(* CoDeSys 2.3 export: ROUNDINGTO5.EXP *)

(* POU 05_Basic_Calc/roundingTo5, ST *)
FUNCTION roundingTo5 : UINT 	(* Функция окргуляет число до ближайшего кратного (5 * order) числа *)
VAR_INPUT
	in_number_u16	: UINT;		(* Число, которое нужно округлить *)
	order				: UINT;		(* Порядок до которого округлять. 1 – до кратного 5ти, 10 – до кратного 50ти, и тд... *)
END_VAR
VAR
	div_part			: REAL;		(* Целое число *)
	aux_num			: UINT;		(* вспомогательная переменная для отслеживания округления до меньшего целого *)
	dec_part			: REAL;		(* десятая часть числа *)
END_VAR
VAR CONSTANT
	LOW_ROUND		: REAL := 0.25;
	HIGH_ROUND		: REAL := 0.75;
END_VAR
IF order < 1 THEN
	roundingTo5 := in_number_u16;
ELSE
	IF order < 10 THEN
		order := 1;
	ELSIF order < 100 THEN
		order := 10;
	ELSIF order < 1000 THEN
		order := 100;
	ELSIF order < 10000 THEN
		order := 1000;
	ELSE
		order := 10000;
	END_IF

	div_part	:= UINT_TO_REAL(in_number_u16) / (order * 10);
	aux_num	:= REAL_TO_UINT(div_part);
	
	IF UINT_TO_REAL(aux_num) > div_part THEN
		aux_num := aux_num - 1;
	END_IF

	dec_part	:= ABS(div_part - UINT_TO_REAL(aux_num));

	IF dec_part >= LOW_ROUND AND  dec_part < HIGH_ROUND THEN
		dec_part := 0.5;
	ELSIF dec_part < LOW_ROUND THEN
		dec_part := 0.0;
	ELSE
		dec_part := 1.0;
	END_IF

	roundingTo5 := (aux_num * (order * 10) + REAL_TO_UINT(dec_part * (order * 10)));
END_IF
END_FUNCTION
